// Mitsubishi GX Works2 project: Class7_Conveyor분류   PLC: Q03UD

PROGRAM MAIN
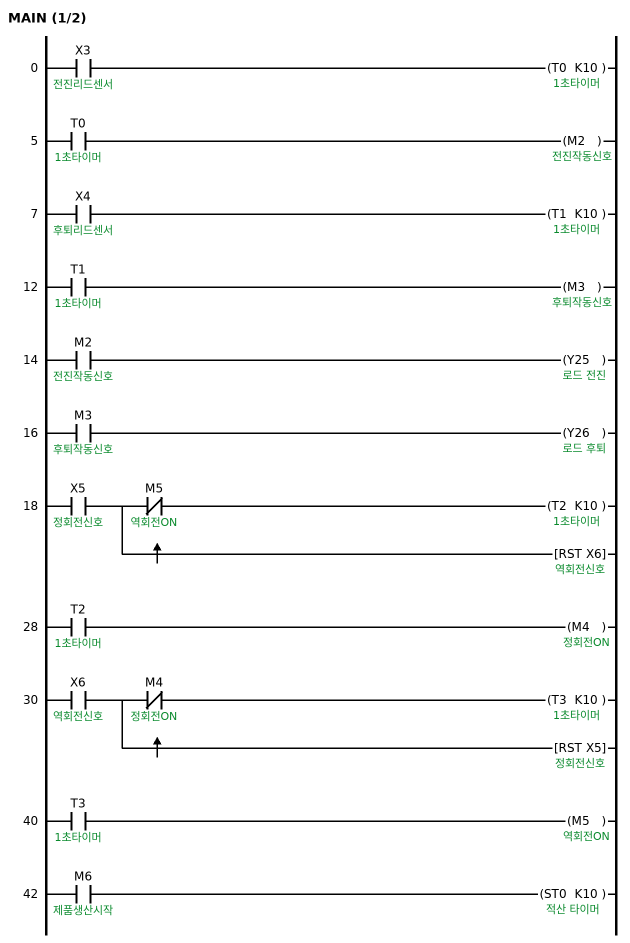
0     LD      X3  ; 전진리드센서
      OUT     T0 K10  ; 1초타이머
5     LD      T0  ; 1초타이머
      OUT     M2  ; 전진작동신호
7     LD      X4  ; 후퇴리드센서
      OUT     T1 K10  ; 1초타이머
12    LD      T1  ; 1초타이머
      OUT     M3  ; 후퇴작동신호
14    LD      M2  ; 전진작동신호
      OUT     Y25  ; 로드 전진
16    LD      M3  ; 후퇴작동신호
      OUT     Y26  ; 로드 후퇴
18    LD      X5  ; 정회전신호
      MPS
      ANI     M5  ; 역회전ON
      OUT     T2 K10  ; 1초타이머
      MPP
      MEP
      RST     X6  ; 역회전신호
28    LD      T2  ; 1초타이머
      OUT     M4  ; 정회전ON
30    LD      X6  ; 역회전신호
      MPS
      ANI     M4  ; 정회전ON
      OUT     T3 K10  ; 1초타이머
      MPP
      MEP
      RST     X5  ; 정회전신호
40    LD      T3  ; 1초타이머
      OUT     M5  ; 역회전ON
42    LD      M6  ; 제품생산시작
      OUT     ST0 K10  ; 적산 타이머
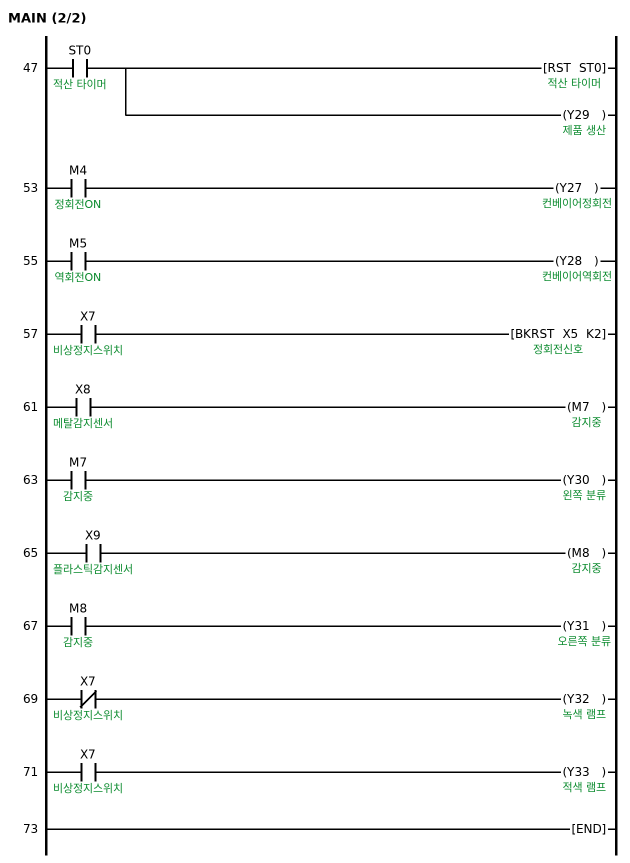
47    LD      ST0  ; 적산 타이머
      RST     ST0  ; 적산 타이머
      OUT     Y29  ; 제품 생산
53    LD      M4  ; 정회전ON
      OUT     Y27  ; 컨베이어정회전
55    LD      M5  ; 역회전ON
      OUT     Y28  ; 컨베이어역회전
57    LD      X7  ; 비상정지스위치
      BKRST   X5 K2
61    LD      X8  ; 메탈감지센서
      OUT     M7  ; 감지중
63    LD      M7  ; 감지중
      OUT     Y30  ; 왼쪽 분류
65    LD      X9  ; 플라스틱감지센서
      OUT     M8  ; 감지중
67    LD      M8  ; 감지중
      OUT     Y31  ; 오른쪽 분류
69    LDI     X7  ; 비상정지스위치
      OUT     Y32  ; 녹색 램프
71    LD      X7  ; 비상정지스위치
      OUT     Y33  ; 적색 램프
73    END
END_PROGRAM

// device comments not shown above
X0  ; 메탈감지센서
X1  ; 플라감지센서
X2  ; 긴급정지버튼
Y0  ; 제품 생산
Y1  ; 왼쪽 분류
Y2  ; 오른쪽분류
Y3  ; 녹색 램프
Y4  ; 적색 램프
M0  ; 감지중
M1  ; 감지중
